(* IEC 61131-3 sources: astools/Data/ASTemplates/Default/Standard Execute FB, 2 files *)

(* ---- __fb_name__Types.typ ---- *)
TYPE
    __fb_name__InternalType :     STRUCT  (*Template of a structure of internal parameters for an execute function block *)
        ExecuteOld : BOOL; (*Variable to detect rising edge on Execute input*)
        Executing : BOOL; (*Executing flag*)
        ParametersValid : BOOL; (*All parameters valid flag*)
        Parameter1 : REAL; (*Internal parameter for computing*)
        Parameter2 : REAL; (*Internal parameter for computing*)
    END_STRUCT;
END_TYPE

(* ---- library.fun ---- *)
FUNCTION_BLOCK __fb_name__ (*FB template for Execute FB*)
    VAR_INPUT
        Execute : BOOL; (*Execute the function block*)
        Parameter1 : REAL; (*Parameter required for computing*)
        Parameter2 : REAL; (*Parameter required for computing*)
        In : REAL; (*Input variable*)
    END_VAR
    VAR_OUTPUT
        Done : BOOL; (*Execute is done*)
        Busy : BOOL; (*Function block is busy*)
        Error : BOOL; (*Indicates an error*)
        StatusID : DINT; (*Status information*)
        Out : REAL; (*Output variable*)
    END_VAR
    VAR
        Internal : __fb_name__InternalType; (*Data for internal use*)
    END_VAR
END_FUNCTION_BLOCK
